Fanuc KAREL source: kt00402.KL

-- PROVISIONAL review KL for V770-1; original PC SHA256 4f794faee5f276e9a5af70e92452d16ca1ccf486d5b5851cef690095c2896fd6
-- Incomplete behavior may be omitted. Consult companion uncertainty JSON. Do not deploy.
PROGRAM KT00402
%NOLOCKGROUP
VAR
  I1 : INTEGER
  R2 : REAL
  OUT : BOOLEAN
BEGIN
  -- UNRESOLVED_PC offsets 5-16; opcodes 2E,23
  -- UNRESOLVED_PC offsets 21-32; opcodes 2E,23
  -- UNRESOLVED_PC offsets 37-59; opcodes 21,21,29,64,29,71,23
  -- UNRESOLVED_PC offsets 64-68; opcodes 7F
END KT00402
